ABB RobotStudio station: myGofa_20220203-161821.rsstn

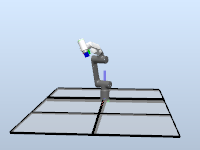
Station myGofa (saved by RobotStudio 21.2.9526.0)
Controller CRB15000_5_95
  mechanical unit ROB_1: CRB15000_5_95__01, 6 joints, base frame (0, 0, 0) mm
Layout (positions relative to the parent item):
  - CRB15000_5_95__01 [mechanism, from Robots\CRB15000_5_95__01.rslib] at (0, 0, 0) mm; joint values [-0.4955, 0.2623, -0.5141, 0.545, 1.6615, -0.8917] (rad or m)
